{attribute 'GeneratedUsingTerminal: EL3204-0000-0017'}
{attribute addProperty BoxType "EL3204-0000-0017"}
{attribute addProperty Id "RTD_Inputs_Channel_1AT %I*RTD_Inputs_Channel_4A3944819RTD_Inputs_Channel_2AT %I*RTD_Inputs_Channel_4A3944819RTD_Inputs_Channel_3AT %I*RTD_Inputs_Channel_4A3944819RTD_Inputs_Channel_4AT %I*RTD_Inputs_Channel_4A3944819WcStateAT %I*WcState_9091E0EB2InfoDataAT %I*InfoData_32EB74EA10"}
{attribute addProperty CRC "1235222566"}
{attribute addProperty Size "48"}
TYPE EL3204_49A00026 EXTENDS EtcSlaveTerminalBase_947E5A46 :
STRUCT
	{attribute addProperty Name "RTD_Inputs_Channel_1"}
	RTD_Inputs_Channel_1 : RTD_Inputs_Channel_4A394481;
	{attribute addProperty Name "RTD_Inputs_Channel_2"}
	RTD_Inputs_Channel_2 : RTD_Inputs_Channel_4A394481;
	{attribute addProperty Name "RTD_Inputs_Channel_3"}
	RTD_Inputs_Channel_3 : RTD_Inputs_Channel_4A394481;
	{attribute addProperty Name "RTD_Inputs_Channel_4"}
	RTD_Inputs_Channel_4 : RTD_Inputs_Channel_4A394481;
	{attribute addProperty Name "WcState"}
	WcState : WcState_9091E0EB;
	{attribute addProperty Name "InfoData"}
	InfoData : InfoData_32EB74EA;
END_STRUCT
END_TYPE

(* stored: Version 1.2.0.0, ProductVersion 3.1.4024.9
   DUT EL3204_49A00026: Id {cd6ae423-cd00-4f0b-8625-5671593d2982} *)
